% RSLogix 500 project I2P Job 22 - Tyler_Vogt.RSS, saved by version 10.00.00.00 %
PROJECT "MLO2B"    % processor: Bul.1763 MicroLogix 1100 Series B %

PROGRAM FILES
  LAD 2   9 rungs

DATA FILES
  O0 OUTPUT  4 elements
  I1 INPUT  6 elements
  S2 STATUS  66 elements
  B3 BINARY  1 elements
  T4 TIMER  2 elements
  C5 COUNTER  1 elements
  R6 CONTROL  1 elements
  N7 INTEGER  1 elements
  F8 FLOAT  1 elements

LADDER 2
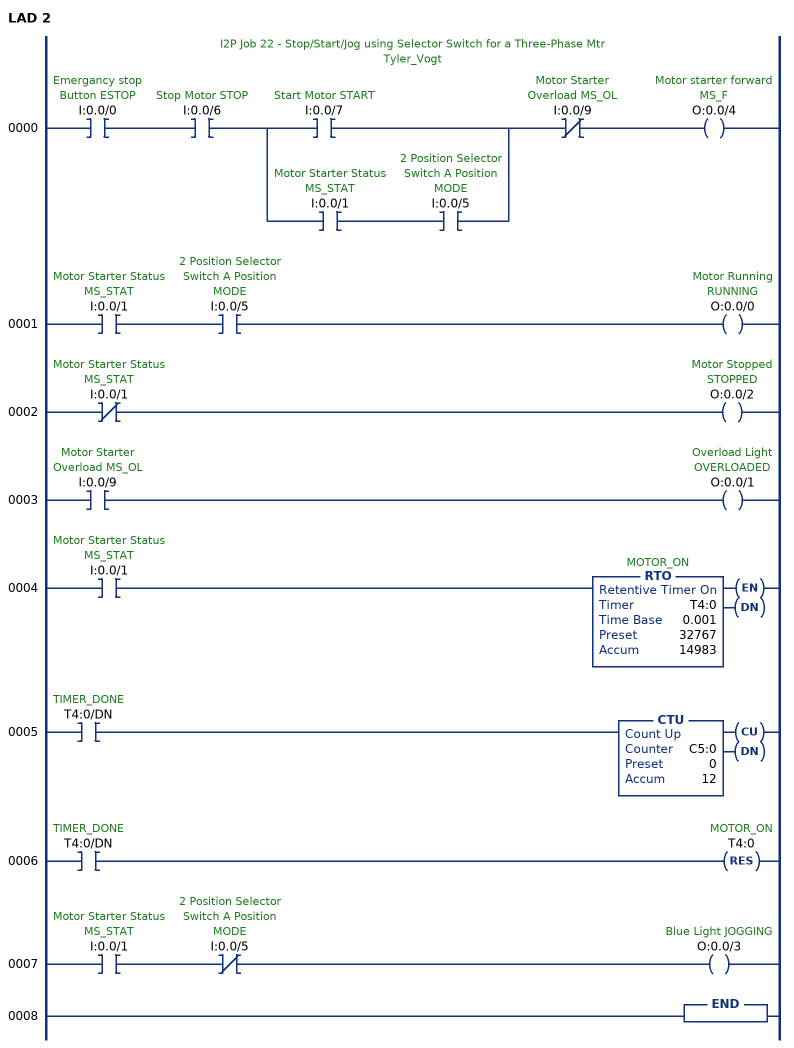
% Rung: 0 %
% I2P Job 22 - Stop/Start/Jog using Selector Switch for a Three-Phase Mtr
% Tyler_Vogt %
SOR XIC I:0.0/0 XIC I:0.0/6 BST XIC I:0.0/7 NXB XIC I:0.0/1 XIC I:0.0/5 BND XIO I:0.0/9 OTE O:0.0/4 EOR
%   I:0.0/0  ESTOP  "Emergancy stop Button" %
%   I:0.0/6  STOP  "Stop Motor" %
%   I:0.0/7  START  "Start Motor" %
%   I:0.0/1  MS_STAT  "Motor Starter Status" %
%   I:0.0/5  MODE  "2 Position Selector Switch A Position" %
%   I:0.0/9  MS_OL  "Motor Starter Overload" %
%   O:0.0/4  MS_F  "Motor starter forward" %
% Rung: 1 %
SOR XIC I:0.0/1 XIC I:0.0/5 OTE O:0.0/0 EOR
%   I:0.0/1  MS_STAT  "Motor Starter Status" %
%   I:0.0/5  MODE  "2 Position Selector Switch A Position" %
%   O:0.0/0  RUNNING  "Motor Running" %
% Rung: 2 %
SOR XIO I:0.0/1 OTE O:0.0/2 EOR
%   I:0.0/1  MS_STAT  "Motor Starter Status" %
%   O:0.0/2  STOPPED  "Motor Stopped" %
% Rung: 3 %
SOR XIC I:0.0/9 OTE O:0.0/1 EOR
%   I:0.0/9  MS_OL  "Motor Starter Overload" %
%   O:0.0/1  OVERLOADED  "Overload Light" %
% Rung: 4 %
SOR XIC I:0.0/1 RTO T4:0 0.001 32767 14983 EOR
%   I:0.0/1  MS_STAT  "Motor Starter Status" %
%   T4:0  MOTOR_ON %
% Rung: 5 %
SOR XIC T4:0/DN CTU C5:0 0 12 EOR
%   T4:0/DN  TIMER_DONE %
% Rung: 6 %
SOR XIC T4:0/DN RES T4:0 EOR
%   T4:0/DN  TIMER_DONE %
%   T4:0  MOTOR_ON %
% Rung: 7 %
SOR XIC I:0.0/1 XIO I:0.0/5 OTE O:0.0/3 EOR
%   I:0.0/1  MS_STAT  "Motor Starter Status" %
%   I:0.0/5  MODE  "2 Position Selector Switch A Position" %
%   O:0.0/3  JOGGING  "Blue Light" %
% Rung: 8 %
SOR END EOR

OTHER DOCUMENTED ADDRESSES
  B3:0/0  AUTO_BIT  "Auto position bit"
  B3:0/1  ON_BIT  "On position bit"
  B3:0/2  FWD_BIT
  B3:0/3  REV_BIT
  B3:0/4  YLW_LT_BIT
  B3:0/5  LAST_REV
  B3:0/6  LAST_FWD
  B3:0/7  STOP_BIT  "Estop and Stop"
  FWD_JOG  "Forward Jog"
  I:0.0/2  DIR_STAT  "Motor Direction Status"
  I:0.0/3  AUTO_POS  "3 Position Selector Switch A Position"
  I:0.0/4  ON  "3 Position Selector Switch B Position"
  I:0.0/8  JOG  "Jog Motor"
  MOTOR  
  O:0.0/5  CR2  "Direction Control Relay"
  T4:0.ACC/0  BLINK_TIMER
  T4:0/EN  TIMER_ENABLED
  T4:0/TT  MOTOR_DELAY_TIMER
  T4:1  FWD_DELAY

DATA TABLE (non-zero values as saved)
DATA B3
% B3:0 % 0X0004
DATA T4
% .PRE .ACC %
% T4:0 % 32767 14983
% T4:1 % 8 0
DATA C5
% .PRE .ACC %
% C5:0 % 0 12
